FUNCTION_BLOCK c_bar (* Composite FB wrapping other FBs *)
  (* Standard: 61499-2; Description: Part of ellipse fitting method, to find c_bar. *)
  (* Version 1.0, 2020-08-19, Candra Wardaya, UGM *)
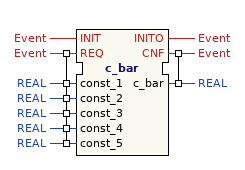
  EVENT_INPUT
    INIT; (* Initialization Request *)
    REQ WITH const_1, const_2, const_3, const_4, const_5; (* Normal Execution Request *)
  END_EVENT
  EVENT_OUTPUT
    INITO; (* Initialization Confirm *)
    CNF WITH c_bar; (* Execution Confirmation *)
  END_EVENT
  VAR_INPUT
    const_1 : REAL; (* Single Real Input *)
    const_2 : REAL; (* Single Real Input *)
    const_3 : REAL; (* Single Real Input *)
    const_4 : REAL; (* Single Real Input *)
    const_5 : REAL; (* Single Real Input *)
  END_VAR
  VAR_OUTPUT
    c_bar : REAL; (* Single Real Output *)
  END_VAR
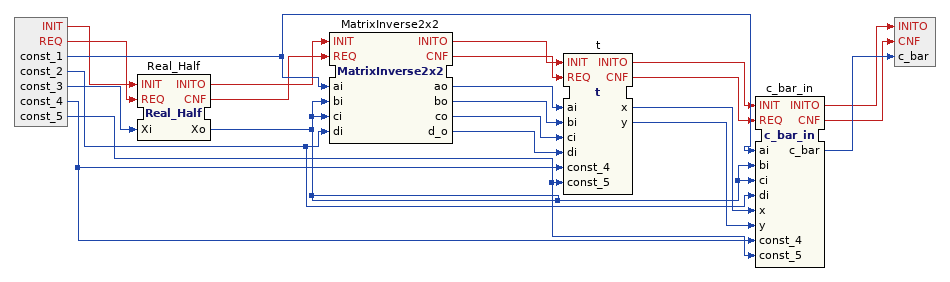
  FBS
    Real_Half : Real_Half;
    MatrixInverse2x2 : MatrixInverse2x2;
    t : t;
    c_bar_in : c_bar_in;
  END_FBS
  EVENT_CONNECTIONS
    REQ TO Real_Half.REQ;
    INIT TO Real_Half.INIT;
    Real_Half.INITO TO MatrixInverse2x2.INIT;
    Real_Half.CNF TO MatrixInverse2x2.REQ;
    MatrixInverse2x2.CNF TO t.REQ;
    MatrixInverse2x2.INITO TO t.INIT;
    t.CNF TO c_bar_in.REQ;
    t.INITO TO c_bar_in.INIT;
    c_bar_in.INITO TO INITO;
    c_bar_in.CNF TO CNF;
  END_CONNECTIONS
  DATA_CONNECTIONS
    Real_Half.Xo TO MatrixInverse2x2.ci;
    Real_Half.Xo TO MatrixInverse2x2.bi;
    const_3 TO Real_Half.Xi;
    const_1 TO MatrixInverse2x2.ai;
    const_2 TO MatrixInverse2x2.di;
    MatrixInverse2x2.ao TO t.ai;
    MatrixInverse2x2.bo TO t.bi;
    MatrixInverse2x2.co TO t.ci;
    MatrixInverse2x2.d_o TO t.di;
    const_4 TO t.const_4;
    const_5 TO t.const_5;
    const_1 TO c_bar_in.ai;
    const_2 TO c_bar_in.di;
    Real_Half.Xo TO c_bar_in.bi;
    Real_Half.Xo TO c_bar_in.ci;
    t.x TO c_bar_in.x;
    t.y TO c_bar_in.y;
    const_4 TO c_bar_in.const_4;
    const_5 TO c_bar_in.const_5;
    c_bar_in.c_bar TO c_bar;
  END_CONNECTIONS
END_FUNCTION_BLOCK
